FUNCTION_BLOCK F_1States_2Algo (* Basic FB with empty ECC *)
  (* Standard: 61499-2 *)
  (* Version 1.0, 2023-09-22, AK124910 *)
  PACKAGE servSeq;
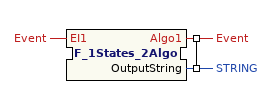
  EVENT_INPUT
    EI1;
  END_EVENT
  EVENT_OUTPUT
    Algo1 WITH OutputString;
  END_EVENT
  VAR_OUTPUT
    OutputString : STRING;
  END_VAR
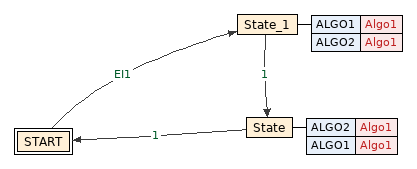
  EC_STATES
    START; (* Initial State *)
    State_1 : ALGO1 -> Algo1, ALGO2 -> Algo1;
    State : ALGO2 -> Algo1, ALGO1 -> Algo1;
  END_STATES
  EC_TRANSITIONS
    START TO State_1 := EI1;
    State_1 TO State := 1;
    State TO START := 1;
  END_TRANSITIONS
  ALGORITHM ALGO1 IN ST:
OutputString := CONCAT(OutputString, 'ALGO1/');
  END_ALGORITHM
  ALGORITHM ALGO2 IN ST:
OutputString := CONCAT(OutputString, 'ALGO2/');
  END_ALGORITHM
  SERVICE external/internal_interface (* Basic FB with empty ECC *)
    SEQUENCE ServiceSequence (* Coverage: 1.0 *) {SET_ATTRIBUTE(StartState, START)}
      external.EI1() -> external.Algo1(OutputString:=STRING#'ALGO1/';) -> external.Algo1(OutputString:=STRING#'ALGO1/ALGO2/';) -> external.Algo1(OutputString:=STRING#'ALGO1/ALGO2/ALGO2/';) -> external.Algo1(OutputString:=STRING#'ALGO1/ALGO2/ALGO2/ALGO1/';);
    END_SEQUENCE
  END_SERVICE
END_FUNCTION_BLOCK
